Staubli VAL3: action_bufferT.pgx

program action_bufferT(ActionItem& x_aAction[] (dimensions=1))
  local num i
  local bool l_bMutex
  local bool l_bTraj
  local num l_nActualStep
  local num l_nIdTask
  local num l_nInstrId
  local num l_nMinus
  local num l_nTask
  local num l_nZero
  local string l_sAction
  local string l_sEmpty
  local string l_sInstrType
begin
  //
  // INIT
  //
  // wait the Task Cycle or simulation has been started
  wait(cycleStatus:bCycle or cycleStatus:bSimulation)
  //
  if x_aAction.iInstr.sType!="" and x_aAction.iInstr.sType!="null"
    // compose the instruction
    // do the action
    x_aAction.nDistance=0
    x_aAction.nMoveId=-1
    x_aAction.nPointId=-1
    call action_do(x_aAction,-1)
  endIf
end
